// TIA Portal V16 export
// export: Created 2022-09-01T14:29:18.7214843Z, ExportSetting WithDefaults, DisplayName Totally Integrated Automation Portal, DisplayVersion V16, DisplayName TIA Portal Version Control Interface, DisplayVersion V16, DisplayName TIA Portal Openness, DisplayVersion V16, DisplayName STEP 7 Professional, DisplayVersion V16, DisplayName STEP 7 Safety, DisplayVersion V16, DisplayName WinCC Advanced, DisplayVersion V16
FUNCTION "Comando_Nível_TK03" : Void   // FC10, LAD
{ S7_Optimized_Access := 'TRUE' }
VERSION : 0.1
// stored: AutoNumber true, IsIECCheckEnabled false, SetENOAutomatically false, UDAEnableTagReadback false
   VAR_INPUT
      Nível_em_Metros : Real;
   END_VAR
   VAR_OUTPUT
      LSH : Bool;
      LSM : Bool;
      LSL : Bool;
   END_VAR
BEGIN

REGION Network 1
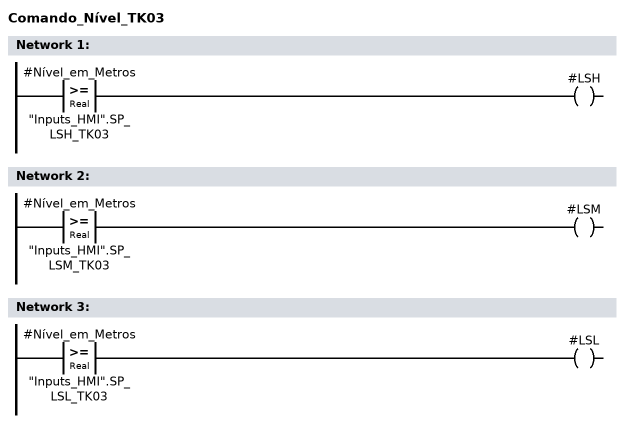
   RUNG wire#powerrail
      { S7_Templates := "SrcType := Real" } GE_Contact(in1 := #Nível_em_Metros, in2 := "Inputs_HMI".SP_LSH_TK03)
      Coil( #LSH )
   END_RUNG
   // the same network as SCL:
   #LSH := #Nível_em_Metros >= "Inputs_HMI".SP_LSH_TK03;
END_REGION

REGION Network 2
   RUNG wire#powerrail
      { S7_Templates := "SrcType := Real" } GE_Contact(in1 := #Nível_em_Metros, in2 := "Inputs_HMI".SP_LSM_TK03)
      Coil( #LSM )
   END_RUNG
   // the same network as SCL:
   #LSM := #Nível_em_Metros >= "Inputs_HMI".SP_LSM_TK03;
END_REGION

REGION Network 3
   RUNG wire#powerrail
      { S7_Templates := "SrcType := Real" } GE_Contact(in1 := #Nível_em_Metros, in2 := "Inputs_HMI".SP_LSL_TK03)
      Coil( #LSL )
   END_RUNG
   // the same network as SCL:
   #LSL := #Nível_em_Metros >= "Inputs_HMI".SP_LSL_TK03;
END_REGION
END_FUNCTION
